// Mitsubishi GX Works2 project: SmartFarmModbusTempDx combin   PLC: FX3U/FX3UC

PROGRAM MAIN
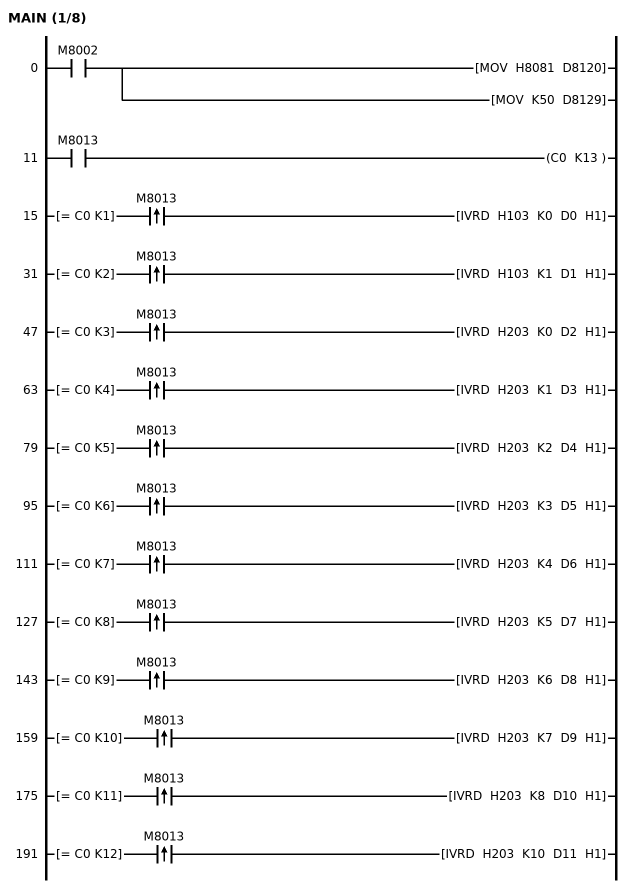
0     LD      M8002
      MOV     H8081 D8120
      MOV     K50 D8129
11    LD      M8013
      OUT     C0 K13
15    LD=     C0 K1
      ANDP    M8013
      IVRD    H103 K0 D0 H1
31    LD=     C0 K2
      ANDP    M8013
      IVRD    H103 K1 D1 H1
47    LD=     C0 K3
      ANDP    M8013
      IVRD    H203 K0 D2 H1
63    LD=     C0 K4
      ANDP    M8013
      IVRD    H203 K1 D3 H1
79    LD=     C0 K5
      ANDP    M8013
      IVRD    H203 K2 D4 H1
95    LD=     C0 K6
      ANDP    M8013
      IVRD    H203 K3 D5 H1
111   LD=     C0 K7
      ANDP    M8013
      IVRD    H203 K4 D6 H1
127   LD=     C0 K8
      ANDP    M8013
      IVRD    H203 K5 D7 H1
143   LD=     C0 K9
      ANDP    M8013
      IVRD    H203 K6 D8 H1
159   LD=     C0 K10
      ANDP    M8013
      IVRD    H203 K7 D9 H1
175   LD=     C0 K11
      ANDP    M8013
      IVRD    H203 K8 D10 H1
191   LD=     C0 K12
      ANDP    M8013
      IVRD    H203 K10 D11 H1
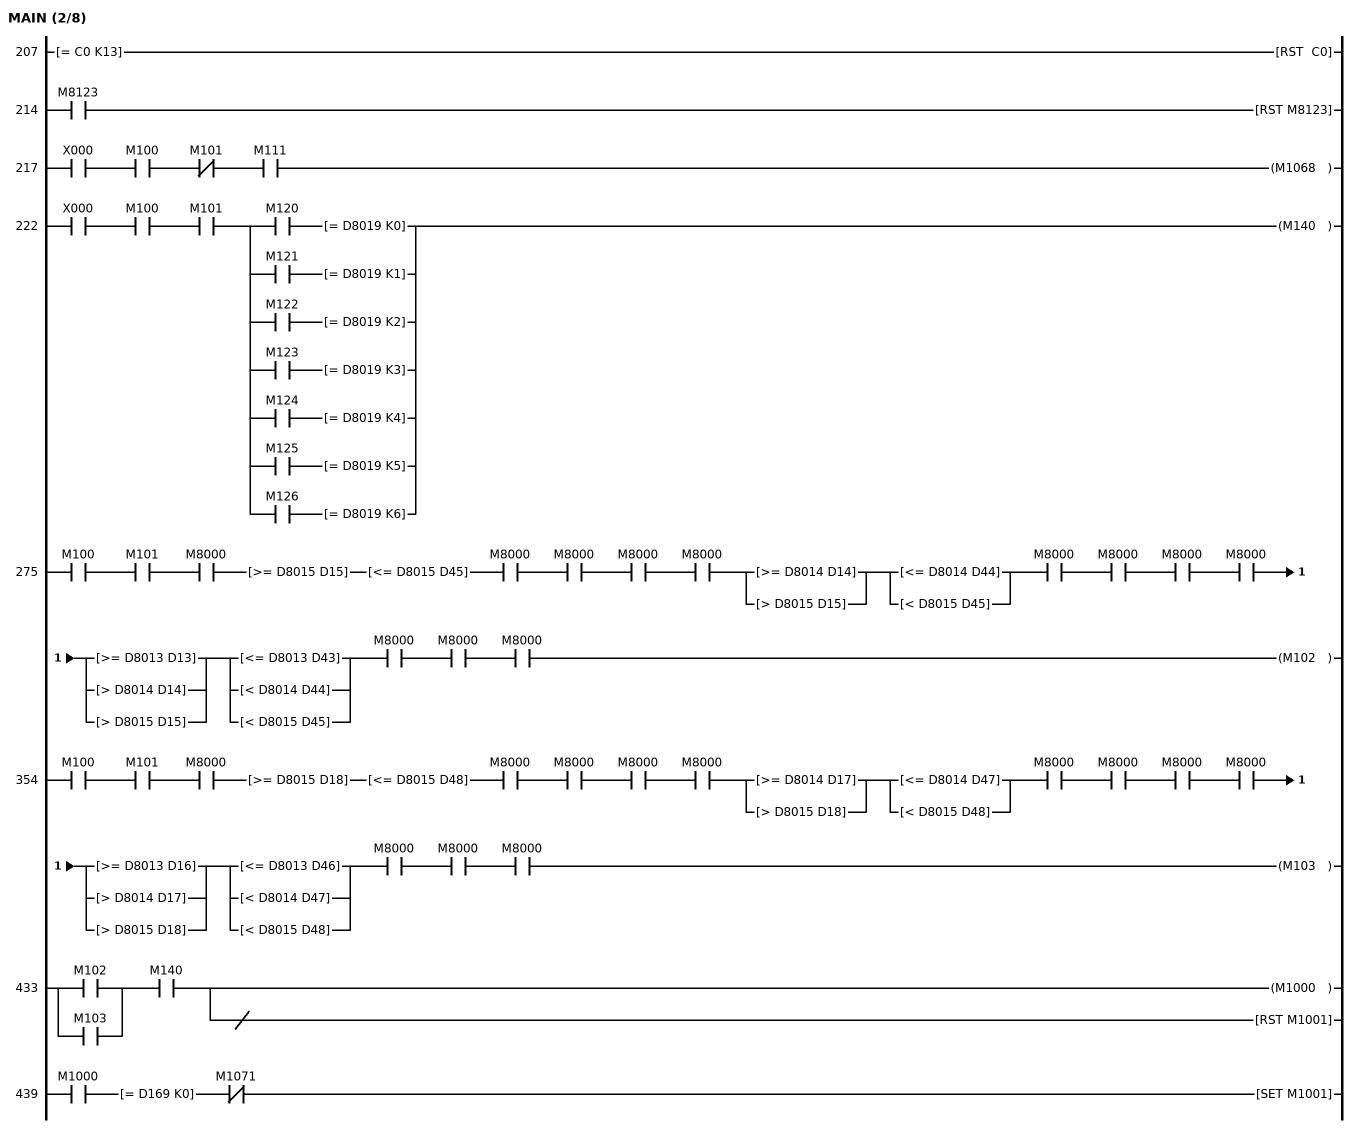
207   LD=     C0 K13
      RST     C0
214   LD      M8123
      RST     M8123
217   LD      X000
      AND     M100
      ANI     M101
      AND     M111
      OUT     M1068
222   LD      X000
      AND     M100
      AND     M101
      LD      M120
      AND=    D8019 K0
      LD      M121
      AND=    D8019 K1
      ORB
      LD      M122
      AND=    D8019 K2
      ORB
      LD      M123
      AND=    D8019 K3
      ORB
      LD      M124
      AND=    D8019 K4
      ORB
      LD      M125
      AND=    D8019 K5
      ORB
      LD      M126
      AND=    D8019 K6
      ORB
      ANB
      OUT     M140
275   LD      M100
      AND     M101
      AND     M8000
      AND>=   D8015 D15
      AND<=   D8015 D45
      AND     M8000
      AND     M8000
      AND     M8000
      AND     M8000
      LD>=    D8014 D14
      OR>     D8015 D15
      ANB
      LD<=    D8014 D44
      OR<     D8015 D45
      ANB
      AND     M8000
      AND     M8000
      AND     M8000
      AND     M8000
      LD>=    D8013 D13
      OR>     D8014 D14
      OR>     D8015 D15
      ANB
      LD<=    D8013 D43
      OR<     D8014 D44
      OR<     D8015 D45
      ANB
      AND     M8000
      AND     M8000
      AND     M8000
      OUT     M102
354   LD      M100
      AND     M101
      AND     M8000
      AND>=   D8015 D18
      AND<=   D8015 D48
      AND     M8000
      AND     M8000
      AND     M8000
      AND     M8000
      LD>=    D8014 D17
      OR>     D8015 D18
      ANB
      LD<=    D8014 D47
      OR<     D8015 D48
      ANB
      AND     M8000
      AND     M8000
      AND     M8000
      AND     M8000
      LD>=    D8013 D16
      OR>     D8014 D17
      OR>     D8015 D18
      ANB
      LD<=    D8013 D46
      OR<     D8014 D47
      OR<     D8015 D48
      ANB
      AND     M8000
      AND     M8000
      AND     M8000
      OUT     M103
433   LD      M102
      OR      M103
      AND     M140
      OUT     M1000
      INV
      RST     M1001
439   LD      M1000
      AND=    D169 K0
      ANI     M1071
      SET     M1001
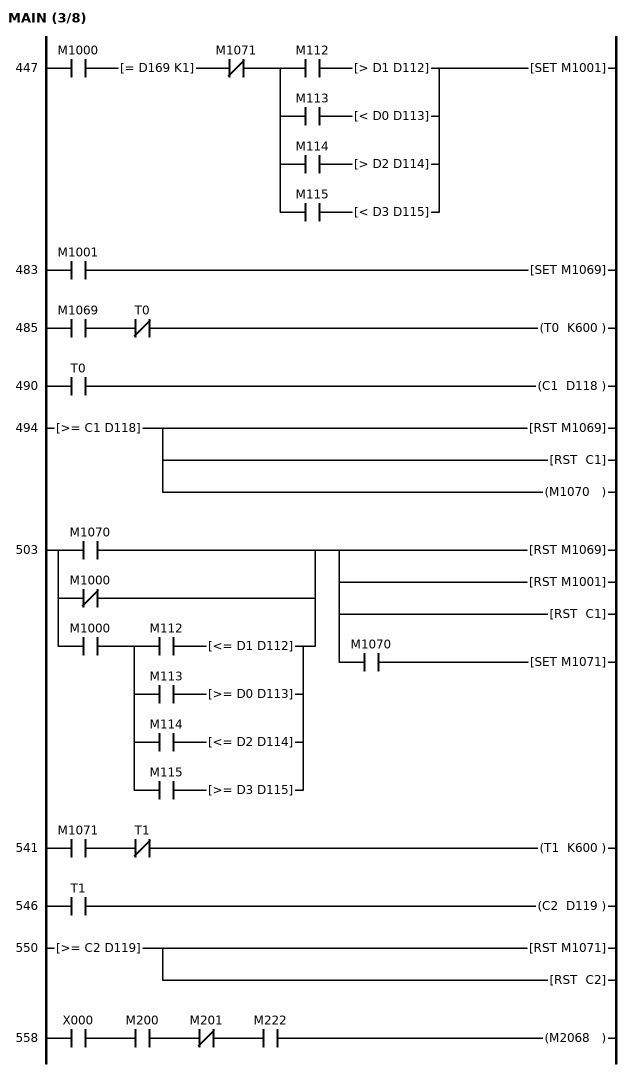
447   LD      M1000
      AND=    D169 K1
      ANI     M1071
      LD      M112
      AND>    D1 D112
      LD      M113
      AND<    D0 D113
      ORB
      LD      M114
      AND>    D2 D114
      ORB
      LD      M115
      AND<    D3 D115
      ORB
      ANB
      SET     M1001
483   LD      M1001
      SET     M1069
485   LD      M1069
      ANI     T0
      OUT     T0 K600
490   LD      T0
      OUT     C1 D118
494   LD>=    C1 D118
      RST     M1069
      RST     C1
      OUT     M1070
503   LD      M1070
      ORI     M1000
      LD      M1000
      LD      M112
      AND<=   D1 D112
      LD      M113
      AND>=   D0 D113
      ORB
      LD      M114
      AND<=   D2 D114
      ORB
      LD      M115
      AND>=   D3 D115
      ORB
      ANB
      ORB
      RST     M1069
      RST     M1001
      RST     C1
      AND     M1070
      SET     M1071
541   LD      M1071
      ANI     T1
      OUT     T1 K600
546   LD      T1
      OUT     C2 D119
550   LD>=    C2 D119
      RST     M1071
      RST     C2
558   LD      X000
      AND     M200
      ANI     M201
      AND     M222
      OUT     M2068
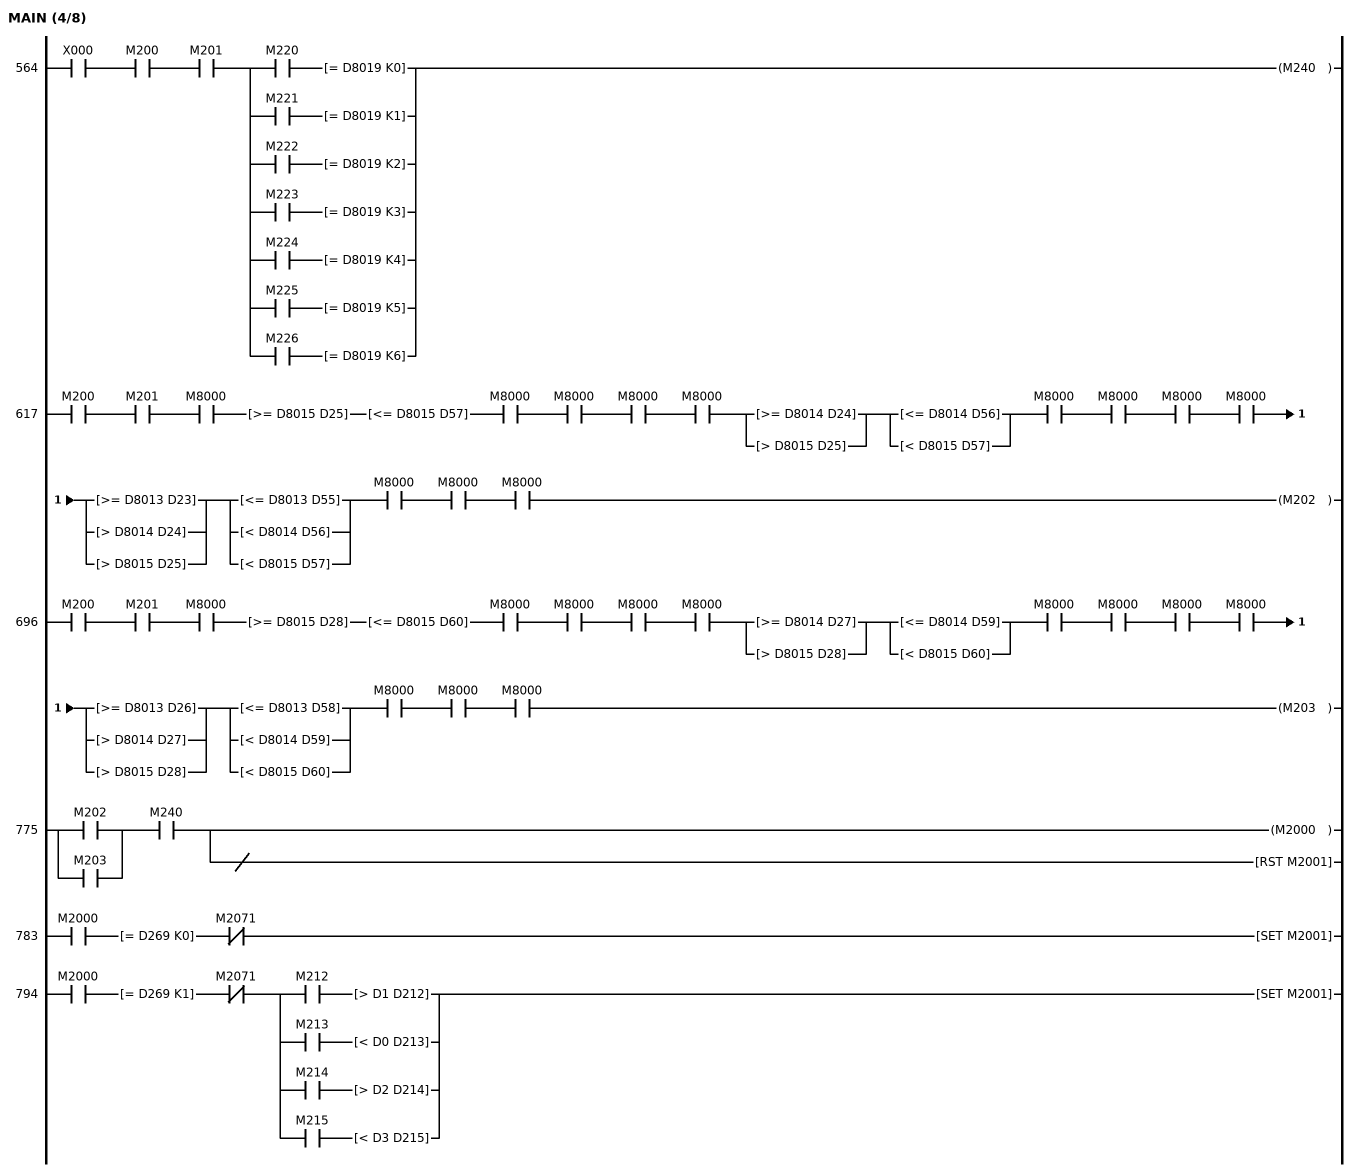
564   LD      X000
      AND     M200
      AND     M201
      LD      M220
      AND=    D8019 K0
      LD      M221
      AND=    D8019 K1
      ORB
      LD      M222
      AND=    D8019 K2
      ORB
      LD      M223
      AND=    D8019 K3
      ORB
      LD      M224
      AND=    D8019 K4
      ORB
      LD      M225
      AND=    D8019 K5
      ORB
      LD      M226
      AND=    D8019 K6
      ORB
      ANB
      OUT     M240
617   LD      M200
      AND     M201
      AND     M8000
      AND>=   D8015 D25
      AND<=   D8015 D57
      AND     M8000
      AND     M8000
      AND     M8000
      AND     M8000
      LD>=    D8014 D24
      OR>     D8015 D25
      ANB
      LD<=    D8014 D56
      OR<     D8015 D57
      ANB
      AND     M8000
      AND     M8000
      AND     M8000
      AND     M8000
      LD>=    D8013 D23
      OR>     D8014 D24
      OR>     D8015 D25
      ANB
      LD<=    D8013 D55
      OR<     D8014 D56
      OR<     D8015 D57
      ANB
      AND     M8000
      AND     M8000
      AND     M8000
      OUT     M202
696   LD      M200
      AND     M201
      AND     M8000
      AND>=   D8015 D28
      AND<=   D8015 D60
      AND     M8000
      AND     M8000
      AND     M8000
      AND     M8000
      LD>=    D8014 D27
      OR>     D8015 D28
      ANB
      LD<=    D8014 D59
      OR<     D8015 D60
      ANB
      AND     M8000
      AND     M8000
      AND     M8000
      AND     M8000
      LD>=    D8013 D26
      OR>     D8014 D27
      OR>     D8015 D28
      ANB
      LD<=    D8013 D58
      OR<     D8014 D59
      OR<     D8015 D60
      ANB
      AND     M8000
      AND     M8000
      AND     M8000
      OUT     M203
775   LD      M202
      OR      M203
      AND     M240
      OUT     M2000
      INV
      RST     M2001
783   LD      M2000
      AND=    D269 K0
      ANI     M2071
      SET     M2001
794   LD      M2000
      AND=    D269 K1
      ANI     M2071
      LD      M212
      AND>    D1 D212
      LD      M213
      AND<    D0 D213
      ORB
      LD      M214
      AND>    D2 D214
      ORB
      LD      M215
      AND<    D3 D215
      ORB
      ANB
      SET     M2001
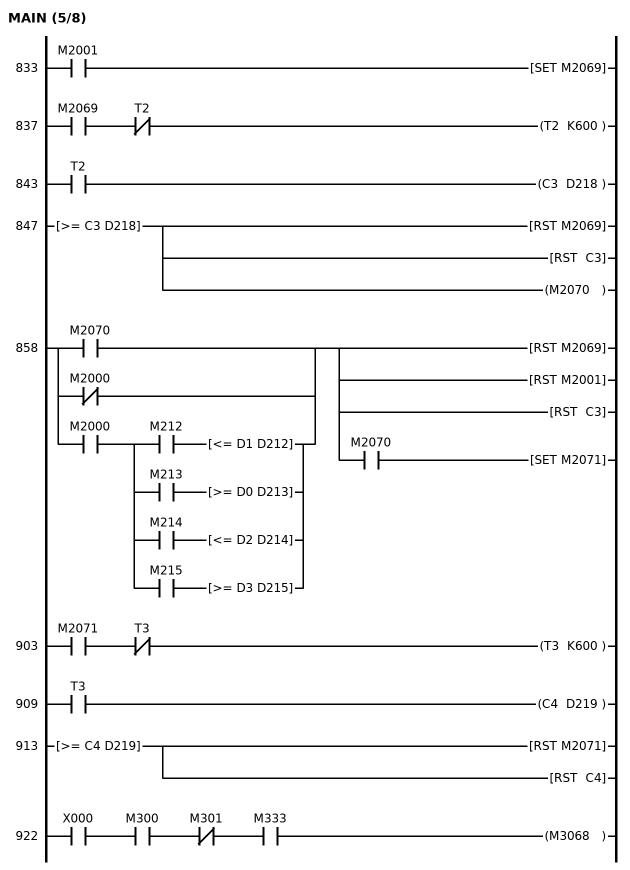
833   LD      M2001
      SET     M2069
837   LD      M2069
      ANI     T2
      OUT     T2 K600
843   LD      T2
      OUT     C3 D218
847   LD>=    C3 D218
      RST     M2069
      RST     C3
      OUT     M2070
858   LD      M2070
      ORI     M2000
      LD      M2000
      LD      M212
      AND<=   D1 D212
      LD      M213
      AND>=   D0 D213
      ORB
      LD      M214
      AND<=   D2 D214
      ORB
      LD      M215
      AND>=   D3 D215
      ORB
      ANB
      ORB
      RST     M2069
      RST     M2001
      RST     C3
      AND     M2070
      SET     M2071
903   LD      M2071
      ANI     T3
      OUT     T3 K600
909   LD      T3
      OUT     C4 D219
913   LD>=    C4 D219
      RST     M2071
      RST     C4
922   LD      X000
      AND     M300
      ANI     M301
      AND     M333
      OUT     M3068
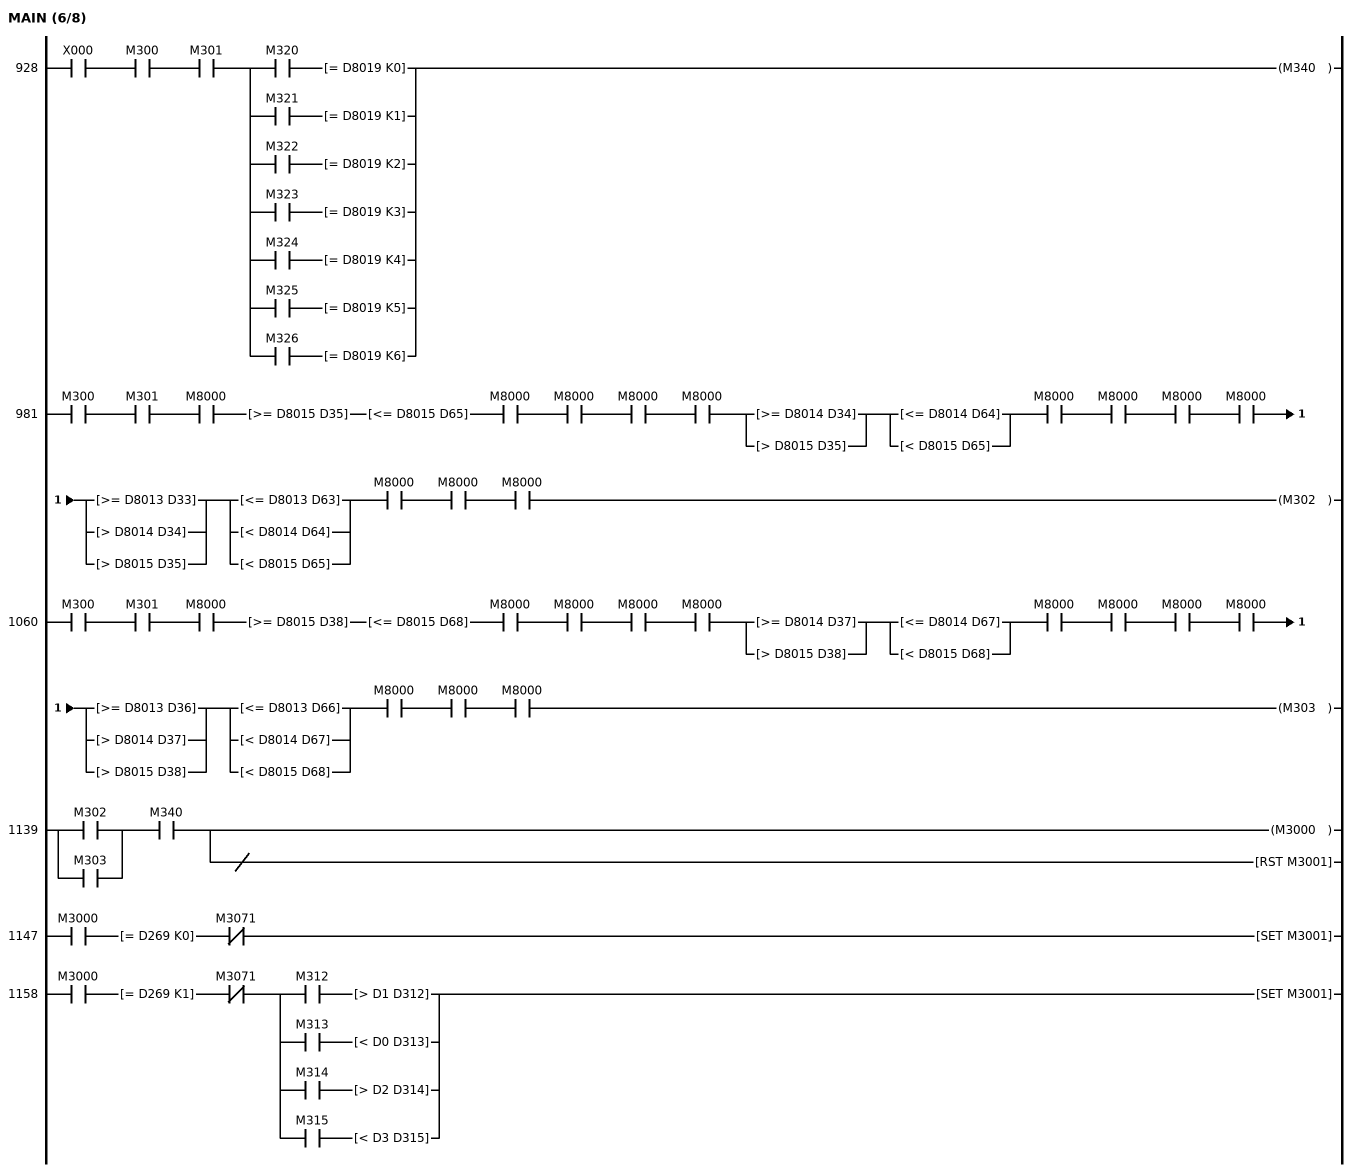
928   LD      X000
      AND     M300
      AND     M301
      LD      M320
      AND=    D8019 K0
      LD      M321
      AND=    D8019 K1
      ORB
      LD      M322
      AND=    D8019 K2
      ORB
      LD      M323
      AND=    D8019 K3
      ORB
      LD      M324
      AND=    D8019 K4
      ORB
      LD      M325
      AND=    D8019 K5
      ORB
      LD      M326
      AND=    D8019 K6
      ORB
      ANB
      OUT     M340
981   LD      M300
      AND     M301
      AND     M8000
      AND>=   D8015 D35
      AND<=   D8015 D65
      AND     M8000
      AND     M8000
      AND     M8000
      AND     M8000
      LD>=    D8014 D34
      OR>     D8015 D35
      ANB
      LD<=    D8014 D64
      OR<     D8015 D65
      ANB
      AND     M8000
      AND     M8000
      AND     M8000
      AND     M8000
      LD>=    D8013 D33
      OR>     D8014 D34
      OR>     D8015 D35
      ANB
      LD<=    D8013 D63
      OR<     D8014 D64
      OR<     D8015 D65
      ANB
      AND     M8000
      AND     M8000
      AND     M8000
      OUT     M302
1060  LD      M300
      AND     M301
      AND     M8000
      AND>=   D8015 D38
      AND<=   D8015 D68
      AND     M8000
      AND     M8000
      AND     M8000
      AND     M8000
      LD>=    D8014 D37
      OR>     D8015 D38
      ANB
      LD<=    D8014 D67
      OR<     D8015 D68
      ANB
      AND     M8000
      AND     M8000
      AND     M8000
      AND     M8000
      LD>=    D8013 D36
      OR>     D8014 D37
      OR>     D8015 D38
      ANB
      LD<=    D8013 D66
      OR<     D8014 D67
      OR<     D8015 D68
      ANB
      AND     M8000
      AND     M8000
      AND     M8000
      OUT     M303
1139  LD      M302
      OR      M303
      AND     M340
      OUT     M3000
      INV
      RST     M3001
1147  LD      M3000
      AND=    D269 K0
      ANI     M3071
      SET     M3001
1158  LD      M3000
      AND=    D269 K1
      ANI     M3071
      LD      M312
      AND>    D1 D312
      LD      M313
      AND<    D0 D313
      ORB
      LD      M314
      AND>    D2 D314
      ORB
      LD      M315
      AND<    D3 D315
      ORB
      ANB
      SET     M3001
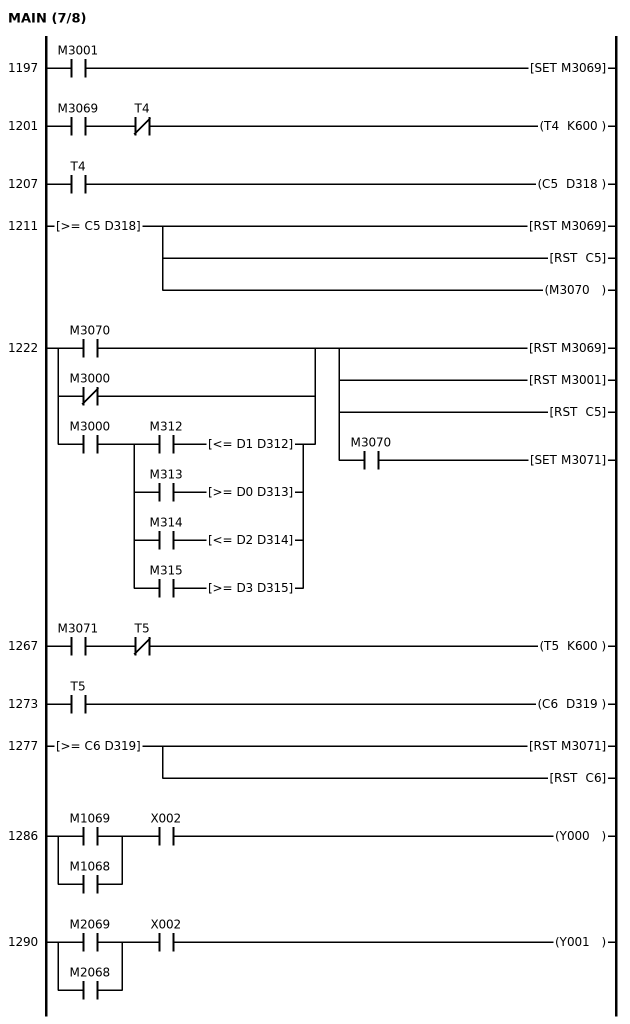
1197  LD      M3001
      SET     M3069
1201  LD      M3069
      ANI     T4
      OUT     T4 K600
1207  LD      T4
      OUT     C5 D318
1211  LD>=    C5 D318
      RST     M3069
      RST     C5
      OUT     M3070
1222  LD      M3070
      ORI     M3000
      LD      M3000
      LD      M312
      AND<=   D1 D312
      LD      M313
      AND>=   D0 D313
      ORB
      LD      M314
      AND<=   D2 D314
      ORB
      LD      M315
      AND>=   D3 D315
      ORB
      ANB
      ORB
      RST     M3069
      RST     M3001
      RST     C5
      AND     M3070
      SET     M3071
1267  LD      M3071
      ANI     T5
      OUT     T5 K600
1273  LD      T5
      OUT     C6 D319
1277  LD>=    C6 D319
      RST     M3071
      RST     C6
1286  LD      M1069
      OR      M1068
      AND     X002
      OUT     Y000
1290  LD      M2069
      OR      M2068
      AND     X002
      OUT     Y001
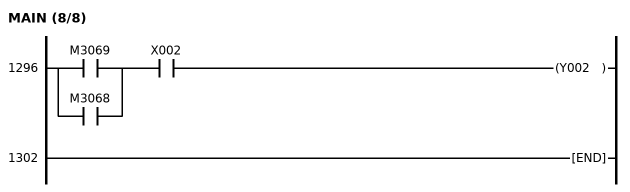
1296  LD      M3069
      OR      M3068
      AND     X002
      OUT     Y002
1302  END
END_PROGRAM
